SUBAPPLICATION AR_SPLIT_2_3 (* Verzweigt 3 unabhaengige AR-Werte auf je 2 Ziele (IN1 auf OUT1a/OUT1b, IN2 auf OUT2a/OUT2b, IN3 auf OUT3a/OUT3b) ueber je einen AR_SPLIT_2. Spart 3x AR_SPLIT_2 als Einzelbausteine, wo mehrere Werte gleichzeitig an zwei unabhaengige Verbraucher verteilt werden muessen (z.B. Schwelle/Totzone/Hysterese an Regel-Logik UND Positions-/Anzeige-Logik, wie in Befuellautomatik). *)
  (* Standard: 61499-2; Description: Copyright (c) 2026 Meisterschulen am Ostbahnhof This program and the accompanying materials are made available under the terms of the Eclipse Public License 2.0 which is available at https://www.eclipse.org/legal/epl-2.0/ SPDX-License-Identifier: EPL-2.0 *)
  (* Version 1.0, 2026-09-27, Franz Höpfinger, Meisterschulen am Ostbahnhof, initial implementation - 3x AR_SPLIT_2 gebuendelt fuer den wiederkehrenden Fall 'mehrere INI-/Referenzwerte gleichzeitig an zwei unabhaengige Verbraucher'. *)
  PACKAGE MyLib::sys;
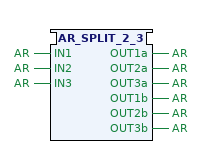
  SOCKETS
    IN1 : adapter::types::unidirectional::AR; (* Wird auf OUT1a und OUT1b verzweigt *)
    IN2 : adapter::types::unidirectional::AR; (* Wird auf OUT2a und OUT2b verzweigt *)
    IN3 : adapter::types::unidirectional::AR; (* Wird auf OUT3a und OUT3b verzweigt *)
  END_SOCKETS
  PLUGS
    OUT1a : adapter::types::unidirectional::AR; (* IN1, erstes Ziel *)
    OUT2a : adapter::types::unidirectional::AR; (* IN2, erstes Ziel *)
    OUT3a : adapter::types::unidirectional::AR; (* IN3, erstes Ziel *)
    OUT1b : adapter::types::unidirectional::AR; (* IN1, zweites Ziel *)
    OUT2b : adapter::types::unidirectional::AR; (* IN2, zweites Ziel *)
    OUT3b : adapter::types::unidirectional::AR; (* IN3, zweites Ziel *)
  END_PLUGS
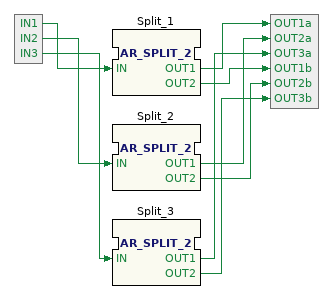
  FBS
    Split_1 : adapter::events::unidirectional::AR_SPLIT_2;
    Split_2 : adapter::events::unidirectional::AR_SPLIT_2;
    Split_3 : adapter::events::unidirectional::AR_SPLIT_2;
  END_FBS
  ADAPTER_CONNECTIONS
    IN1 TO Split_1.IN;
    Split_1.OUT1 TO OUT1a;
    Split_1.OUT2 TO OUT1b;
    IN2 TO Split_2.IN;
    Split_2.OUT1 TO OUT2a;
    Split_2.OUT2 TO OUT2b;
    IN3 TO Split_3.IN;
    Split_3.OUT1 TO OUT3a;
    Split_3.OUT2 TO OUT3b;
  END_CONNECTIONS
END_SUBAPPLICATION
